DATA_BLOCK "dbArchiveParTank"
{ S7_Optimized_Access := 'TRUE' }
VERSION : 0.8
"fbArchiveParTank"

BEGIN

END_DATA_BLOCK

